(*20-34 Fehler Mit Quittierung*)
OfMeldung[uiI_FehlerId_Riem1+20]:= strIO_GHdshk_Riem1.b_MMaxLaufzeit_AufBahn;
OfMeldung[uiI_FehlerId_Riem1+21]:= strIO_GHdshk_Riem1.b_MMaxLaufzeit_VonBahn;
OfMeldung[uiI_FehlerId_Riem1+22]:= strIO_GHdshk_Riem1.b_MBahnNichtAufFoerderhoehe;
OfMeldung[uiI_FehlerId_Riem1+23]:= FALSE;
OfMeldung[uiI_FehlerId_Riem1+24]:= FALSE;
OfMeldung[uiI_FehlerId_Riem1+25]:= strIO_GHdshk_Riem1.b_MBahnBelegt_KeineDaten;
OfMeldung[uiI_FehlerId_Riem1+26]:= strIO_GHdshk_Riem1.b_MBahnFrei_Daten;
OfMeldung[uiI_FehlerId_Riem1+27]:= strIO_GHdshk_Riem1.b_MFehlerRegisterimpuls;
OfMeldung[uiI_FehlerId_Riem1+28]:= strIO_GHdshk_Riem1.b_MKeineFreigabe_FahrtInGrund;
OfMeldung[uiI_FehlerId_Riem1+29]:= strIO_GHdshk_Riem1.b_MTeilNichtFreigegeben;
OfMeldung[uiI_FehlerId_Riem1+30]:= strIO_GHdshk_Riem1.b_MFehlerSkalierung;
OfMeldung[uiI_FehlerId_Riem1+31]:= FALSE;
OfMeldung[uiI_FehlerId_Riem1+32]:= FALSE;
OfMeldung[uiI_FehlerId_Riem1+33]:= FALSE;
OfMeldung[uiI_FehlerId_Riem1+34]:= FALSE;

(*35-49 Fehler ohne Quittierung*)
OfMeldung[uiI_FehlerId_Riem1+35]:= FALSE;
OfMeldung[uiI_FehlerId_Riem1+36]:= FALSE;
OfMeldung[uiI_FehlerId_Riem1+37]:= FALSE;
OfMeldung[uiI_FehlerId_Riem1+38]:= FALSE;	
OfMeldung[uiI_FehlerId_Riem1+39]:= FALSE;
OfMeldung[uiI_FehlerId_Riem1+40]:= FALSE;
OfMeldung[uiI_FehlerId_Riem1+41]:= FALSE;
OfMeldung[uiI_FehlerId_Riem1+42]:= FALSE;
OfMeldung[uiI_FehlerId_Riem1+43]:= FALSE;
OfMeldung[uiI_FehlerId_Riem1+44]:= FALSE;
OfMeldung[uiI_FehlerId_Riem1+45]:= FALSE;
OfMeldung[uiI_FehlerId_Riem1+46]:= FALSE;
OfMeldung[uiI_FehlerId_Riem1+47]:= FALSE;
OfMeldung[uiI_FehlerId_Riem1+48]:= FALSE;
OfMeldung[uiI_FehlerId_Riem1+49]:= FALSE;

strIO_Stoerungen.bStoerungAntriebe:=
	strIO_Stoerungen.bStoerungAntriebe
	OR	F_MeldungAktiv( Von:= uiI_FehlerId_Riem1, Bis:= uiI_FehlerId_Riem1 + 4, Anzahl:= 0, Raster:= 0 );

strIO_Stoerungen.bAbsoluterStop:=
	strIO_Stoerungen.bAbsoluterStop
	OR	F_MeldungAktiv( Von:= uiI_FehlerId_Riem1 + 5, Bis:= uiI_FehlerId_Riem1 + 9, Anzahl:= 0, Raster:= 0 );

strIO_Stoerungen.bBedingterStop:=
	strIO_Stoerungen.bBedingterStop
	OR	F_MeldungAktiv( Von:= uiI_FehlerId_Riem1 + 10, Bis:= uiI_FehlerId_Riem1 + 19, Anzahl:= 0, Raster:= 0 );

strIO_Stoerungen.bFehlerMitQuittung:=
	strIO_Stoerungen.bFehlerMitQuittung
	OR	F_MeldungAktiv( Von:= uiI_FehlerId_Riem1 + 20, Bis:= uiI_FehlerId_Riem1 + 34, Anzahl:= 0, Raster:= 0 );

strIO_Stoerungen.bFehlerOhneQuittung:=
	strIO_Stoerungen.bFehlerOhneQuittung
	OR	F_MeldungAktiv( Von:= uiI_FehlerId_Riem1 + 35, Bis:= uiI_FehlerId_Riem1 + 49, Anzahl:= 0, Raster:= 0 );
END_ACTION

ACTION Z_Meldungen_Riem2:
(*----------------------------------------------------------------------------------------------------------------------------------*)
(*----------------------------------------------------------------------------------------------------------------------------------*)
(*                Meldungen																		*)
(*----------------------------------------------------------------------------------------------------------------------------------*)
(*----------------------------------------------------------------------------------------------------------------------------------*)

(*0-4 Störung Antriebe*)
OfMeldung[uiI_FehlerId_Riem2+0]:= strIO_GHdshk_Riem2.b_MStoerungAntrieb;
OfMeldung[uiI_FehlerId_Riem2+1]:= FALSE;
OfMeldung[uiI_FehlerId_Riem2+2]:= FALSE;
OfMeldung[uiI_FehlerId_Riem2+3]:= FALSE;
OfMeldung[uiI_FehlerId_Riem2+4]:= FALSE;

(*5-9 Fehler Absoluter Stop*)
OfMeldung[uiI_FehlerId_Riem2+5]:= FALSE;
OfMeldung[uiI_FehlerId_Riem2+6]:= FALSE;
OfMeldung[uiI_FehlerId_Riem2+7]:= FALSE;
OfMeldung[uiI_FehlerId_Riem2+8]:= FALSE;
OfMeldung[uiI_FehlerId_Riem2+9]:= FALSE;

(*10-19 Fehler Bedingter Stop*)
OfMeldung[uiI_FehlerId_Riem2+10]:= fbRampe_Riem2.bQ_Error
						AND 	fbRampe_Riem2.uiQ_ErrorNumber = 100;
OfMeldung[uiI_FehlerId_Riem2+11]:= fbRampe_Riem2.bQ_Error
						AND 	fbRampe_Riem2.uiQ_ErrorNumber = 101;
OfMeldung[uiI_FehlerId_Riem2+12]:= fbRampe_Riem2.bQ_Error
						AND 	fbRampe_Riem2.uiQ_ErrorNumber = 102;
OfMeldung[uiI_FehlerId_Riem2+13]:= fbRampe_Riem2.bQ_Error
						AND 	fbRampe_Riem2.uiQ_ErrorNumber = 103;
OfMeldung[uiI_FehlerId_Riem2+14]:= fbRampe_Riem2.bQ_Error
						AND 	fbRampe_Riem2.uiQ_ErrorNumber = 104;
OfMeldung[uiI_FehlerId_Riem2+15]:= fbRampe_Riem2.bQ_Error
						AND 	fbRampe_Riem2.uiQ_ErrorNumber = 105;
OfMeldung[uiI_FehlerId_Riem2+16]:= FALSE;
OfMeldung[uiI_FehlerId_Riem2+17]:= FALSE;
OfMeldung[uiI_FehlerId_Riem2+18]:= FALSE;

IF	uiI_AxId_Riem2 > 0
THEN
	OfMeldung[uiI_FehlerId_Riem2+19]:= NOT AxFrNcGeeicht[uiI_AxId_Riem2];
ELSE
	OfMeldung[uiI_FehlerId_Riem2+19]:= FALSE;
END_IF;

(*20-34 Fehler Mit Quittierung*)
OfMeldung[uiI_FehlerId_Riem2+20]:= strIO_GHdshk_Riem2.b_MMaxLaufzeit_AufBahn;
OfMeldung[uiI_FehlerId_Riem2+21]:= strIO_GHdshk_Riem2.b_MMaxLaufzeit_VonBahn;
OfMeldung[uiI_FehlerId_Riem2+22]:= strIO_GHdshk_Riem2.b_MBahnNichtAufFoerderhoehe;
OfMeldung[uiI_FehlerId_Riem2+23]:= FALSE;
OfMeldung[uiI_FehlerId_Riem2+24]:= FALSE;
OfMeldung[uiI_FehlerId_Riem2+25]:= strIO_GHdshk_Riem2.b_MBahnBelegt_KeineDaten;
OfMeldung[uiI_FehlerId_Riem2+26]:= strIO_GHdshk_Riem2.b_MBahnFrei_Daten;
OfMeldung[uiI_FehlerId_Riem2+27]:= strIO_GHdshk_Riem2.b_MFehlerRegisterimpuls;
OfMeldung[uiI_FehlerId_Riem2+28]:= strIO_GHdshk_Riem2.b_MKeineFreigabe_FahrtInGrund;
OfMeldung[uiI_FehlerId_Riem2+29]:= strIO_GHdshk_Riem2.b_MTeilNichtFreigegeben;
OfMeldung[uiI_FehlerId_Riem2+30]:= strIO_GHdshk_Riem2.b_MFehlerSkalierung;
OfMeldung[uiI_FehlerId_Riem2+31]:= FALSE;
OfMeldung[uiI_FehlerId_Riem2+32]:= FALSE;
OfMeldung[uiI_FehlerId_Riem2+33]:= FALSE;
OfMeldung[uiI_FehlerId_Riem2+34]:= FALSE;

(*35-49 Fehler ohne Quittierung*)
OfMeldung[uiI_FehlerId_Riem2+35]:= FALSE;
OfMeldung[uiI_FehlerId_Riem2+36]:= FALSE;
OfMeldung[uiI_FehlerId_Riem2+37]:= FALSE;
OfMeldung[uiI_FehlerId_Riem2+38]:= FALSE;	
OfMeldung[uiI_FehlerId_Riem2+39]:= FALSE;
OfMeldung[uiI_FehlerId_Riem2+40]:= FALSE;
OfMeldung[uiI_FehlerId_Riem2+41]:= FALSE;
OfMeldung[uiI_FehlerId_Riem2+42]:= FALSE;
OfMeldung[uiI_FehlerId_Riem2+43]:= FALSE;
OfMeldung[uiI_FehlerId_Riem2+44]:= FALSE;
OfMeldung[uiI_FehlerId_Riem2+45]:= FALSE;
OfMeldung[uiI_FehlerId_Riem2+46]:= FALSE;
OfMeldung[uiI_FehlerId_Riem2+47]:= FALSE;
OfMeldung[uiI_FehlerId_Riem2+48]:= FALSE;
OfMeldung[uiI_FehlerId_Riem2+49]:= FALSE;

strIO_Stoerungen.bStoerungAntriebe:=
	strIO_Stoerungen.bStoerungAntriebe
	OR	F_MeldungAktiv( Von:= uiI_FehlerId_Riem2, Bis:= uiI_FehlerId_Riem2 + 4, Anzahl:= 0, Raster:= 0 );

strIO_Stoerungen.bAbsoluterStop:=
	strIO_Stoerungen.bAbsoluterStop
	OR	F_MeldungAktiv( Von:= uiI_FehlerId_Riem2 + 5, Bis:= uiI_FehlerId_Riem2 + 9, Anzahl:= 0, Raster:= 0 );

strIO_Stoerungen.bBedingterStop:=
	strIO_Stoerungen.bBedingterStop
	OR	F_MeldungAktiv( Von:= uiI_FehlerId_Riem2 + 10, Bis:= uiI_FehlerId_Riem2 + 19, Anzahl:= 0, Raster:= 0 );

strIO_Stoerungen.bFehlerMitQuittung:=
	strIO_Stoerungen.bFehlerMitQuittung
	OR	F_MeldungAktiv( Von:= uiI_FehlerId_Riem2 + 20, Bis:= uiI_FehlerId_Riem2 + 34, Anzahl:= 0, Raster:= 0 );

strIO_Stoerungen.bFehlerOhneQuittung:=
	strIO_Stoerungen.bFehlerOhneQuittung
	OR	F_MeldungAktiv( Von:= uiI_FehlerId_Riem2 + 35, Bis:= uiI_FehlerId_Riem2 + 49, Anzahl:= 0, Raster:= 0 );
END_ACTION

ACTION Z_Meldungen_Roll1:
(*----------------------------------------------------------------------------------------------------------------------------------*)
(*----------------------------------------------------------------------------------------------------------------------------------*)
(*                Meldungen																		*)
(*----------------------------------------------------------------------------------------------------------------------------------*)
(*----------------------------------------------------------------------------------------------------------------------------------*)

(*0-4 Störung Antriebe*)
OfMeldung[uiI_FehlerId_Roll1+0]:= strIO_GHdshk_Roll1.b_MStoerungAntrieb;
OfMeldung[uiI_FehlerId_Roll1+1]:= FALSE;
OfMeldung[uiI_FehlerId_Roll1+2]:= FALSE;
OfMeldung[uiI_FehlerId_Roll1+3]:= FALSE;
OfMeldung[uiI_FehlerId_Roll1+4]:= FALSE;

(*5-9 Fehler Absoluter Stop*)
OfMeldung[uiI_FehlerId_Roll1+5]:= FALSE;
OfMeldung[uiI_FehlerId_Roll1+6]:= FALSE;
OfMeldung[uiI_FehlerId_Roll1+7]:= FALSE;
OfMeldung[uiI_FehlerId_Roll1+8]:= FALSE;
OfMeldung[uiI_FehlerId_Roll1+9]:= FALSE;

(*10-19 Fehler Bedingter Stop*)
OfMeldung[uiI_FehlerId_Roll1+10]:= fbRampe_Roll1.bQ_Error
						AND 	fbRampe_Roll1.uiQ_ErrorNumber = 100;
OfMeldung[uiI_FehlerId_Roll1+11]:= fbRampe_Roll1.bQ_Error
						AND 	fbRampe_Roll1.uiQ_ErrorNumber = 101;
OfMeldung[uiI_FehlerId_Roll1+12]:= fbRampe_Roll1.bQ_Error
						AND 	fbRampe_Roll1.uiQ_ErrorNumber = 102;
OfMeldung[uiI_FehlerId_Roll1+13]:= fbRampe_Roll1.bQ_Error
						AND 	fbRampe_Roll1.uiQ_ErrorNumber = 103;
OfMeldung[uiI_FehlerId_Roll1+14]:= fbRampe_Roll1.bQ_Error
						AND 	fbRampe_Roll1.uiQ_ErrorNumber = 104;
OfMeldung[uiI_FehlerId_Roll1+15]:= fbRampe_Roll1.bQ_Error
						AND 	fbRampe_Roll1.uiQ_ErrorNumber = 105;
OfMeldung[uiI_FehlerId_Roll1+16]:= FALSE;
OfMeldung[uiI_FehlerId_Roll1+17]:= FALSE;
OfMeldung[uiI_FehlerId_Roll1+18]:= FALSE;

IF	uiI_AxId_Roll1 > 0
THEN
	OfMeldung[uiI_FehlerId_Roll1+19]:= NOT AxFrNcGeeicht[uiI_AxId_Roll1];
ELSE
	OfMeldung[uiI_FehlerId_Roll1+19]:= FALSE;
END_IF;

(*20-34 Fehler Mit Quittierung*)
OfMeldung[uiI_FehlerId_Roll1+20]:= strIO_GHdshk_Roll1.b_MMaxLaufzeit_AufBahn;
OfMeldung[uiI_FehlerId_Roll1+21]:= strIO_GHdshk_Roll1.b_MMaxLaufzeit_VonBahn;
OfMeldung[uiI_FehlerId_Roll1+22]:= strIO_GHdshk_Roll1.b_MBahnNichtAufFoerderhoehe;
OfMeldung[uiI_FehlerId_Roll1+23]:= FALSE;
OfMeldung[uiI_FehlerId_Roll1+24]:= FALSE;
OfMeldung[uiI_FehlerId_Roll1+25]:= strIO_GHdshk_Roll1.b_MBahnBelegt_KeineDaten;
OfMeldung[uiI_FehlerId_Roll1+26]:= strIO_GHdshk_Roll1.b_MBahnFrei_Daten;
OfMeldung[uiI_FehlerId_Roll1+27]:= strIO_GHdshk_Roll1.b_MFehlerRegisterimpuls;
OfMeldung[uiI_FehlerId_Roll1+28]:= strIO_GHdshk_Roll1.b_MKeineFreigabe_FahrtInGrund;
OfMeldung[uiI_FehlerId_Roll1+29]:= strIO_GHdshk_Roll1.b_MTeilNichtFreigegeben;
OfMeldung[uiI_FehlerId_Roll1+30]:= strIO_GHdshk_Roll1.b_MFehlerSkalierung;
OfMeldung[uiI_FehlerId_Roll1+31]:= FALSE;
OfMeldung[uiI_FehlerId_Roll1+32]:= FALSE;
OfMeldung[uiI_FehlerId_Roll1+33]:= FALSE;
OfMeldung[uiI_FehlerId_Roll1+34]:= FALSE;

(*35-49 Fehler ohne Quittierung*)
OfMeldung[uiI_FehlerId_Roll1+35]:= FALSE;
OfMeldung[uiI_FehlerId_Roll1+36]:= FALSE;
OfMeldung[uiI_FehlerId_Roll1+37]:= FALSE;
OfMeldung[uiI_FehlerId_Roll1+38]:= FALSE;	
OfMeldung[uiI_FehlerId_Roll1+39]:= FALSE;
OfMeldung[uiI_FehlerId_Roll1+40]:= FALSE;
OfMeldung[uiI_FehlerId_Roll1+41]:= FALSE;
OfMeldung[uiI_FehlerId_Roll1+42]:= FALSE;
OfMeldung[uiI_FehlerId_Roll1+43]:= FALSE;
OfMeldung[uiI_FehlerId_Roll1+44]:= FALSE;
OfMeldung[uiI_FehlerId_Roll1+45]:= FALSE;
OfMeldung[uiI_FehlerId_Roll1+46]:= FALSE;
OfMeldung[uiI_FehlerId_Roll1+47]:= FALSE;
OfMeldung[uiI_FehlerId_Roll1+48]:= FALSE;
OfMeldung[uiI_FehlerId_Roll1+49]:= FALSE;

strIO_Stoerungen.bStoerungAntriebe:=
	strIO_Stoerungen.bStoerungAntriebe
	OR	F_MeldungAktiv( Von:= uiI_FehlerId_Roll1, Bis:= uiI_FehlerId_Roll1 + 4, Anzahl:= 0, Raster:= 0 );

strIO_Stoerungen.bAbsoluterStop:=
	strIO_Stoerungen.bAbsoluterStop
	OR	F_MeldungAktiv( Von:= uiI_FehlerId_Roll1 + 5, Bis:= uiI_FehlerId_Roll1 + 9, Anzahl:= 0, Raster:= 0 );

strIO_Stoerungen.bBedingterStop:=
	strIO_Stoerungen.bBedingterStop
	OR	F_MeldungAktiv( Von:= uiI_FehlerId_Roll1 + 10, Bis:= uiI_FehlerId_Roll1 + 19, Anzahl:= 0, Raster:= 0 );

strIO_Stoerungen.bFehlerMitQuittung:=
	strIO_Stoerungen.bFehlerMitQuittung
	OR	F_MeldungAktiv( Von:= uiI_FehlerId_Roll1 + 20, Bis:= uiI_FehlerId_Roll1 + 34, Anzahl:= 0, Raster:= 0 );

strIO_Stoerungen.bFehlerOhneQuittung:=
	strIO_Stoerungen.bFehlerOhneQuittung
	OR	F_MeldungAktiv( Von:= uiI_FehlerId_Roll1 + 35, Bis:= uiI_FehlerId_Roll1 + 49, Anzahl:= 0, Raster:= 0 );
END_ACTION

END_FUNCTION_BLOCK

(* stored: Version 1.1.0.1, ProductVersion 3.1.4024.12
   POU FB_Bahnhardware_Winkel_1Roll_2Riem: Id {0cd5184b-11ea-463f-a5a9-a1bf9a1e8341}, SpecialFunc None
   Action A_Bahnmodi_Riem1: Id {2fff4163-e318-40b7-a96e-915cb6bb6784}
   Action A_Bahnmodi_Riem2: Id {9c64007d-6ae3-488d-bd4f-fe7f101304d0}
   Action A_Bahnmodi_Roll1: Id {2379256b-2152-4e3f-b162-ff5260b434b9}
   Action B_Zeiten_Rampen_Speed_Riem1: Id {68765d1f-874c-486b-b3bb-de155e95d036}
   Action B_Zeiten_Rampen_Speed_Riem2: Id {296ba5ac-8fab-4b7f-bcbd-52b1ea0576f6}
   Action B_Zeiten_Rampen_Speed_Roll1: Id {6b686fdb-f809-4974-9d48-5fb95f183e63}
   Action C_Eingaenge_Riem1: Id {401a30e8-e0a7-420f-948e-0f587b8f4262}
   Action C_Eingaenge_Riem2: Id {5180db05-ba1c-4794-83d1-e0e347ef8621}
   Action C_Eingaenge_Roll1: Id {96816c7f-875e-437f-bcdc-bf314ad47f9f}
   Action D_Bahnjob_Riem1: Id {0fb96135-b193-43ee-87c8-786aa83003ce}
   Action D_Bahnjob_Riem2: Id {c144b625-c825-4599-a791-973f113114b1}
   Action D_Bahnjob_Roll1: Id {f197565d-b29a-4841-9297-4b9afbee23f1}
   Action E_Ausgaenge_Hub: Id {a9db11da-a553-4d3c-8901-ace94c453a7a}
   Action E_Ausgaenge_Riem1: Id {4bf71f4f-bbac-4148-ac7c-55aefdc24bb1}
   Action E_Ausgaenge_Riem2: Id {eb0f9453-6053-4c22-95f9-26675c356495}
   Action E_Ausgaenge_Roll1: Id {10edfa06-3159-46ca-aecb-841c62febae4}
   Action F_Positionierung_Riem1: Id {2dd52e60-e480-4bdd-a712-fd40bc5bee57}
   Action F_Positionierung_Riem2: Id {e2b11baa-2698-4b03-96e4-a66c39cf0f43}
   Action F_Positionierung_Roll1: Id {fb856b48-ff16-477b-8c69-d172ae4a4359}
   Action G_Protokoll_Riem1: Id {e83e8443-8baf-4260-a743-54f63d768f5e}
   Action G_Protokoll_Riem2: Id {69b4c2a0-3d5b-4de4-b905-723afe3e3530}
   Action G_Protokoll_Roll1: Id {2fcd7de6-9313-485c-ae78-ebf38e59606e}
   Action H_Funktionsauswertung_Riem1: Id {d37820db-df25-457e-9a48-988286c48e25}
   Action H_Funktionsauswertung_Riem2: Id {42220141-85fe-4200-b30e-ec617e9e1784}
   Action H_Funktionsauswertung_Roll1: Id {bcab9cc0-1d45-4734-af7c-b2071f3678a8}
   Action H_Funktionsauswertung_Verriegelung: Id {11f1d799-06a3-48cc-9d1a-319ca90c7bbf}
   Action I_TrEstati_Diagnose: Id {64a32da4-2f26-47bc-9dd0-a91ba21b8649}
   Action Y_Struktur_Riem1: Id {1f3f4e8f-84bf-4e6f-80a0-3f7061275725}
   Action Y_Struktur_Riem2: Id {bd52e485-01b8-4021-9a21-1910782f4b44}
   Action Y_Struktur_Roll1: Id {de73598c-2fd8-439a-b44d-b5eaab3ca7c3}
   Action Z_Meldungen_Riem1: Id {582af093-c6e3-47ec-8a4e-4570155b47dd}
   Action Z_Meldungen_Riem2: Id {41597f38-74ea-47cb-a99b-bef50e80316b}
   Action Z_Meldungen_Roll1: Id {e8fb436d-dd1e-4e9d-89e1-6145f1002133} *)
